# EPICS autosave request: ARAmpApp/Db/aramp_settings_50W1000DM2.req
# This file specifies which PVs of the corresponding database should be saved.

# Enable
$(P)$(R)Enbl-Sel

# Gain
$(P)$(R)Gain-SP
